TYPE OutputBase_10CEE7DE :
STRUCT
END_STRUCT
END_TYPE

(* stored: Version 1.2.0.0, ProductVersion 3.1.4024.9
   DUT OutputBase_10CEE7DE: Id {5e8cff71-5610-404e-8a23-8b9567a78e32} *)
